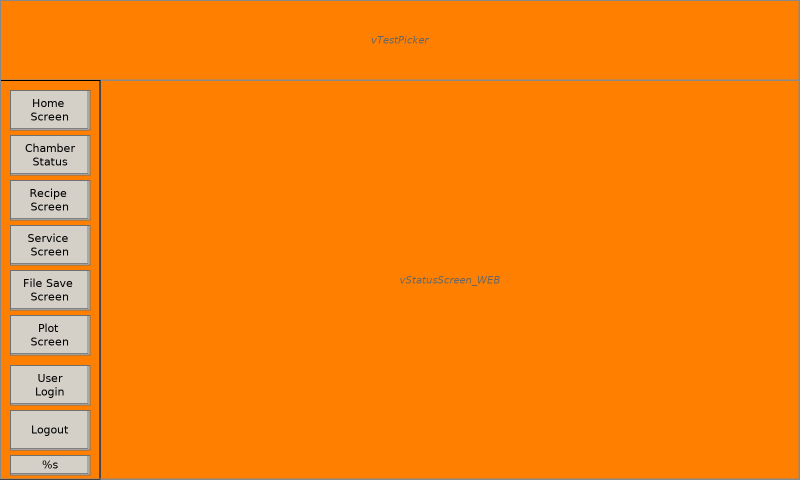
VISUALIZATION vMainScreen_WEB  // 800x480
VAR_IN_OUT
	arChamber : 	ARRAY[0..3] OF fbChamber;
	arParams :   ARRAY[0..3] OF stParamsChamber;
	arControl :   ARRAY[0..3] OF stControl;
	arTestParams : ARRAY[0..3] OF stTestParams;
END_VAR
VAR
	iActualChamber : INT;
	bLogin			: BOOL;
END_VAR
    Frame (0,0 800x80)
        shows vTestPicker(iCompressorPick := arParams[iActualChamber].iCompresorType, iTestType := arControl[iActualChamber].iSetTest, iActualChamber := iActualChamber, arControl := arControl)
    Frame (100,80 700x400)
        shows vStatusScreen_WEB(arChamber := arChamber, arParams := arParams, arControl := arControl)
        shows vRecipe(fbChamber := arChamber[iActualChamber], stChamberTestParams := arTestParams[arParams[iActualChamber].iCompresorType])
        shows vService(fbChamber := arChamber[iActualChamber], stParams := arParams[iActualChamber])
        shows vFileSave(fbChamber := arChamber[iActualChamber], stParams := arParams[iActualChamber])
        shows vPlotScreen(stControl := arControl[iActualChamber], fbChamber := arChamber[iActualChamber])
        shows vStatusScreen_v2_WEB(arChamber := arChamber[iActualChamber], arParams := arParams[iActualChamber], arControl := arControl[iActualChamber])
    Rectangle (0,80 100x400)
    Button (10,90 80x40), "Home Screen"
        OnMouseClick: FrameSelectionChange Selection=SelectedFrame=4e77f9b9-a257-46d1-860a-d32039bd6f78, GlobSel=IndExpr=4, AssignDir=vMainScreen.GenElemInst_5, AssignType=Directly, SelType=Locally
    Button (10,180 80x40), "Recipe Screen"
        OnMouseClick: FrameSelectionChange Selection=SelectedFrame=4e77f9b9-a257-46d1-860a-d32039bd6f78, Selection=1, GlobSel=IndExpr=1, AssignDir=vMainScreen.GenElemInst_5, AssignType=Directly, SelType=Locally
    Button (10,270 80x40), "File Save Screen"
        OnMouseClick: FrameSelectionChange Selection=SelectedFrame=4e77f9b9-a257-46d1-860a-d32039bd6f78, Selection=3, GlobSel=IndExpr=3, AssignDir=vMainScreen.GenElemInst_5, AssignType=Directly, SelType=Locally
    Button (10,225 80x40), "Service Screen"
        OnMouseClick: FrameSelectionChange Selection=SelectedFrame=4e77f9b9-a257-46d1-860a-d32039bd6f78, Selection=2, GlobSel=IndExpr=2, AssignDir=vMainScreen.GenElemInst_5, AssignType=Directly, SelType=Locally
    Button (10,315 80x40), "Plot Screen"
        OnMouseClick: FrameSelectionChange Selection=SelectedFrame=4e77f9b9-a257-46d1-860a-d32039bd6f78, Selection=4, GlobSel=IndExpr=4, AssignDir=vMainScreen.GenElemInst_5, AssignType=Directly, SelType=Locally
    Button (10,365 80x40), "User Login", pressed state: bLogin
        OnMouseClick: VisuUserMgmt Type=Login
    Button (10,410 80x40), "Logout", pressed state: bLogin
        OnMouseClick: VisuUserMgmt Type=Logout
    Button (10,455 80x20), "%s", text variable: Visu_Globals.CurrentUserGroupName, pressed state: bLogin
    Button (10,135 80x40), "Chamber Status"
        OnMouseClick: FrameSelectionChange Selection=SelectedFrame=4e77f9b9-a257-46d1-860a-d32039bd6f78, Selection=5, GlobSel=IndExpr=4, AssignDir=vMainScreen.GenElemInst_5, AssignType=Directly, SelType=Locally
END_VISUALIZATION

(* stored: Version 1.1.0.1, ProductVersion 3.1.4024.12
   Visu vMainScreen_WEB: Id {55049803-85d7-4fd3-aa87-e4fa1ff836f0} *)
